PROGRAM MAIN
VAR
END_VAR

END_PROGRAM

(* stored: Version 1.1.0.1
   POU MAIN: Id {dc5d3262-2c75-40be-bcf4-e3452be8a2b3} *)
